Yaskawa INFORM job: 001-S1_HOME.JBI

/JOB
//NAME 001-S1_HOME
//POS
///NPOS 0,0,1,0,0,0
///TOOL 0
///POSTYPE PULSE
///PULSE
EC00000=0
//INST
///DATE 2025/08/21 14:01
///ATTR SC,RW
///GROUP1 ST1
NOP
MOVJ EC00000 VJ=100.00
END
